FUNCTION_BLOCK FB_Object_Template_SFC
VAR_INPUT
	// Control variables
	Execute: BOOL;
	Ack: BOOL;
	SFCReset: BOOL; 
	SFCPause: BOOL;
	IC: BOOL;
	// Physical variables
END_VAR
VAR_OUTPUT
	//Control variables
	Ready: BOOL;
	Done: BOOL;
	//Physical Variables
END_VAR
VAR
END_VAR

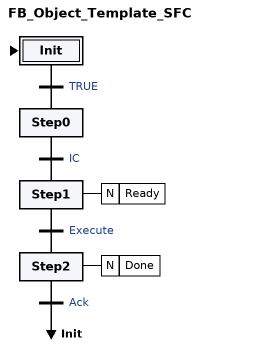
INITIAL_STEP Init:
END_STEP
TRANSITION FROM Init TO Step0
    := TRUE;
END_TRANSITION
STEP Step0:
END_STEP
TRANSITION FROM Step0 TO Step1
    := IC;
END_TRANSITION
STEP Step1:
    Ready(N);
END_STEP
TRANSITION FROM Step1 TO Step2
    := Execute;
END_TRANSITION
STEP Step2:
    Done(N);
END_STEP
TRANSITION FROM Step2 TO Init
    := Ack;
END_TRANSITION

END_FUNCTION_BLOCK

(* stored: Version 1.1.0.1, ProductVersion 3.1.4024.6
   POU FB_Object_Template_SFC: Id {7aa37bff-8033-453f-8a18-c21a3dd6f3b9}, SpecialFunc None *)
